FUNCTION_BLOCK HardWireSequence
VAR
	ready : BOOL;
	contUp : BOOL;
	contDown : BOOL;
	target : REAL := -1;
	
	hardWiredSlider : TeknicHardWire;
END_VAR

hardWiredSlider.bEnable := TRUE;

IF NOT ready THEN
	ready := hardWiredSlider.homingSequence();
	RETURN;
END_IF

hardWiredSlider.stop();
IF contUp THEN
	hardWiredSlider.moveContinuous(direction := MC_Positive_Direction);
	contDown := FALSE;
END_IF

IF contDown THEN
	hardWiredSlider.moveContinuous(direction := MC_Negative_Direction);
	contUp := FALSE;
END_IF


IF target >= 0 THEN
	hardWiredSlider.moveAbsolute(newTarget := target);
	//target := 0;
END_IF


IF hardWiredSlider.innerLimit THEN
	contDown := FALSE;
END_IF
IF hardWiredSlider.home THEN
	contUp := FALSE;
END_IF


hardWiredSlider();

END_FUNCTION_BLOCK

(* stored: Version 1.1.0.1, ProductVersion 3.1.4024.11
   POU HardWireSequence: Id {feb96b66-ea9e-4005-aefa-8ed7917004cc}, SpecialFunc None *)
